FUNCTION_BLOCK XOR (* Logical XOR *)
  (* Standard: 61499-2 *)
  (* Version 1.0, 02.01.2011, gsha041, UoA, Initial Version *)
  (* Compiler header: package fb.rt.UoA; *)
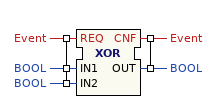
  EVENT_INPUT
    REQ WITH IN1, IN2; (* Normal Execution Request *)
  END_EVENT
  EVENT_OUTPUT
    CNF WITH OUT; (* Execution Confirmation *)
  END_EVENT
  VAR_INPUT
    IN1 : BOOL; (* Argument *)
    IN2 : BOOL; (* Argument *)
  END_VAR
  VAR_OUTPUT
    OUT : BOOL; (* Result: IN1 XOR IN2 XOR ... *)
  END_VAR
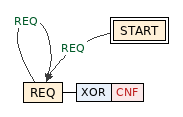
  EC_STATES
    START; (* Initial State *)
    REQ : XOR -> CNF; (* Normal execution *)
  END_STATES
  EC_TRANSITIONS
    START TO REQ := REQ;
    REQ TO REQ := REQ;
  END_TRANSITIONS
  ALGORITHM XOR IN ST: (* Normally executed algorithm *)
OUT := true;
IF IN1 AND IN2 THEN
 OUT := false;
 ELSEIF NOT IN1 AND NOT IN2 THEN OUT := false; END_IF;
  END_ALGORITHM
END_FUNCTION_BLOCK
